(* Logix 5000 project; controller APM Emulate 5570 rev 30.12; software revision 30.00 *)

TASK MainTask (continuous, watchdog 500 ms) : MainProgram

MODULES
   Local : Emulate 5570 (ICP 2, rev 30.12)
      I_O1 : vendor 1 type 0 code 15 (ICP 3, rev 1.1, Output RPI 150 ms)
      I_O2 : vendor 1 type 0 code 15 (ICP 4, rev 1.1, Output RPI 150 ms)
END_MODULES

PROGRAM MainProgram   (* main routine MainRoutine *)
VAR
   CT_ACT_C050 : BOOL;
   CT_ACT_C051 : BOOL;
   CT_ACT_C052 : BOOL;
   CT_ACT_C053 : BOOL;
   CT_ACT_C054 : BOOL;
   CT_ACT_C055 : BOOL;
   CT_ACT_C056 : BOOL;
   CT_ACT_C260 : BOOL;
   CT_ACT_C261 : BOOL;
   CT_ACT_C262 : BOOL;
   CT_ACT_C263 : BOOL;
   CT_ACT_C264 : BOOL;
   CT_ACT_C265 : BOOL;
   CT_ACT_C266 : BOOL;
   CT_ACT_HOM : BOOL;
   CT_ACT_MSP0 : BOOL;
   CT_ACT_MSP1 : BOOL;
   CT_ACT_STP : BOOL;
   CT_ACT_VER0 : BOOL;
   CT_ACT_VER1 : BOOL;
   CT_ACT_VER2 : BOOL;
   CT_CA_AVC : BOOL;
   CT_CA_RET : BOOL;
   CT_CC_AVC : BOOL;
   CT_CC_RET : BOOL;
   CT_CP_AVC : BOOL;
   CT_CP_RET : BOOL;
   CT_DIS : INT;
   CT_OK : BOOL;
   CT_PBT_ESTP : ALIAS FOR Local:4:I.Data[1].0;
   CT_PBT_STA : ALIAS FOR Local:4:I.Data[1].1;
   CT_PBT_STP : ALIAS FOR Local:4:I.Data[1].2;
   CT_SEN_AAV : ALIAS FOR Local:4:I.Data[1].4;
   CT_SEN_ARE : ALIAS FOR Local:4:I.Data[1].3;
   CT_SEN_CAV : ALIAS FOR Local:4:I.Data[1].6;
   CT_SEN_CRE : ALIAS FOR Local:4:I.Data[1].5;
   CT_SEN_M05 : ALIAS FOR Local:4:I.Data[1].11;
   CT_SEN_M26 : ALIAS FOR Local:4:I.Data[1].12;
   CT_SEN_MAT : ALIAS FOR Local:4:I.Data[1].9;
   CT_SEN_PAV : ALIAS FOR Local:4:I.Data[1].8;
   CT_SEN_PRE : ALIAS FOR Local:4:I.Data[1].7;
   CT_SEQ_C05 : BOOL;
   CT_SEQ_C26 : BOOL;
   CT_SEQ_MSP : BOOL;
   CT_SEQ_VER : BOOL;
   MAIN_ACTIVE : BOOL;
   MAIN_PBT_ESTP : ALIAS FOR Local:3:I.Data[1].0;
   MAIN_PBT_STA : ALIAS FOR Local:3:I.Data[1].1;
   PNT_ACT_0 : BOOL;
   PNT_ACT_1 : BOOL;
   PNT_ACT_2 : BOOL;
   PNT_ACT_3 : BOOL;
   PNT_ACT_4 : BOOL;
   PNT_ACT_HOM : BOOL;
   PNT_MTA_AVC : BOOL;
   PNT_MTA_RET : BOOL;
   PNT_MTA_STP : BOOL;
   PNT_MTB_AVC : BOOL;
   PNT_MTB_RET : BOOL;
   PNT_MTB_STP : BOOL;
   PNT_MTC_AVC : BOOL;
   PNT_MTC_RET : BOOL;
   PNT_MTC_STP : BOOL;
   PNT_PBT_HOM : ALIAS FOR Local:3:I.Data[1].10;
   PNT_PBT_STA : ALIAS FOR Local:3:I.Data[1].11;
   PNT_PBT_STP : ALIAS FOR Local:3:I.Data[1].12;
   PNT_SEN_1 : ALIAS FOR Local:3:I.Data[1].13;
   PNT_SEN_2 : ALIAS FOR Local:3:I.Data[1].14;
   PNT_SEN_3 : ALIAS FOR Local:3:I.Data[1].15;
   PNT_SEN_4 : ALIAS FOR Local:3:I.Data[1].16;
   PNT_SEN_5 : ALIAS FOR Local:3:I.Data[1].17;
   PNT_SEN_6 : ALIAS FOR Local:3:I.Data[1].18;
   PNT_SEN_7 : ALIAS FOR Local:3:I.Data[1].19;
   PNT_TM1 : TIMER := (PRE := 2000);
   test : BOOL;
END_VAR

ROUTINE Corte_actions   (* ladder *)
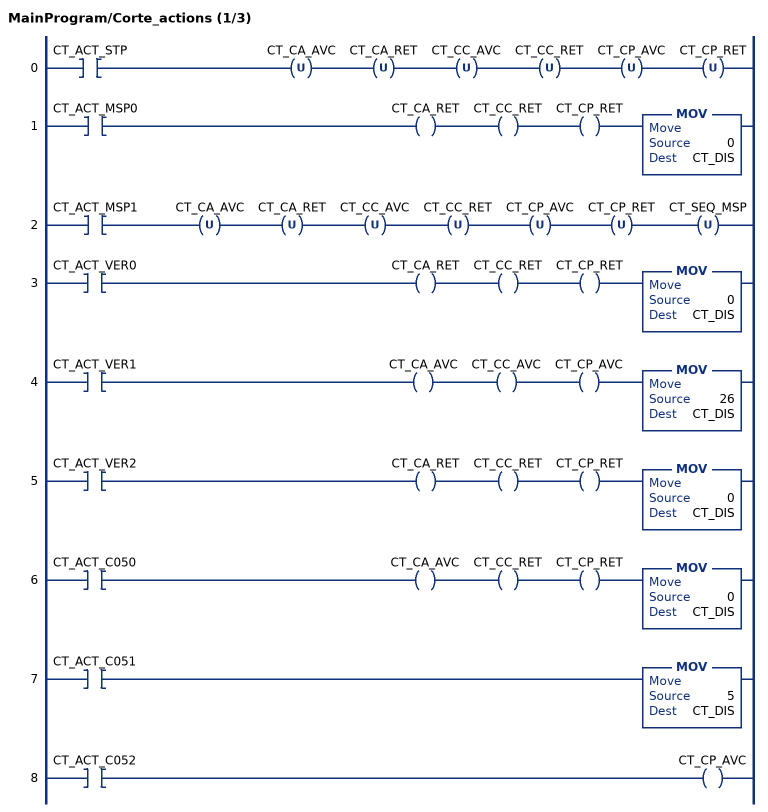
   0: XIC(CT_ACT_STP)OTU(CT_CA_AVC)OTU(CT_CA_RET)OTU(CT_CC_AVC)OTU(CT_CC_RET)OTU(CT_CP_AVC)OTU(CT_CP_RET);
   1: XIC(CT_ACT_MSP0)OTE(CT_CA_RET)OTE(CT_CC_RET)OTE(CT_CP_RET)MOV(0,CT_DIS);
   2: XIC(CT_ACT_MSP1)OTU(CT_CA_AVC)OTU(CT_CA_RET)OTU(CT_CC_AVC)OTU(CT_CC_RET)OTU(CT_CP_AVC)OTU(CT_CP_RET)OTU(CT_SEQ_MSP);
   3: XIC(CT_ACT_VER0)OTE(CT_CA_RET)OTE(CT_CC_RET)OTE(CT_CP_RET)MOV(0,CT_DIS);
   4: XIC(CT_ACT_VER1)OTE(CT_CA_AVC)OTE(CT_CC_AVC)OTE(CT_CP_AVC)MOV(26,CT_DIS);
   5: XIC(CT_ACT_VER2)OTE(CT_CA_RET)OTE(CT_CC_RET)OTE(CT_CP_RET)MOV(0,CT_DIS);
   6: XIC(CT_ACT_C050)OTE(CT_CA_AVC)OTE(CT_CC_RET)OTE(CT_CP_RET)MOV(0,CT_DIS);
   7: XIC(CT_ACT_C051)MOV(5,CT_DIS);
   8: XIC(CT_ACT_C052)OTE(CT_CP_AVC);
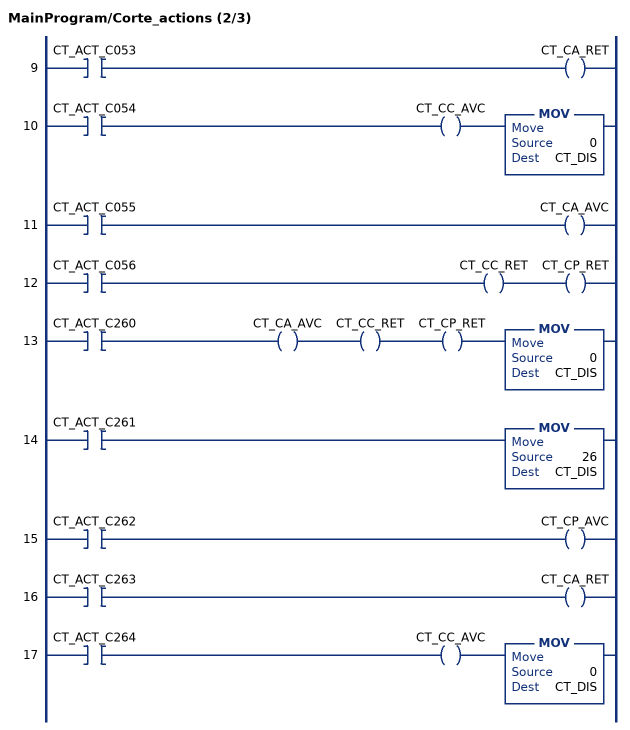
   9: XIC(CT_ACT_C053)OTE(CT_CA_RET);
   10: XIC(CT_ACT_C054)OTE(CT_CC_AVC)MOV(0,CT_DIS);
   11: XIC(CT_ACT_C055)OTE(CT_CA_AVC);
   12: XIC(CT_ACT_C056)OTE(CT_CC_RET)OTE(CT_CP_RET);
   13: XIC(CT_ACT_C260)OTE(CT_CA_AVC)OTE(CT_CC_RET)OTE(CT_CP_RET)MOV(0,CT_DIS);
   14: XIC(CT_ACT_C261)MOV(26,CT_DIS);
   15: XIC(CT_ACT_C262)OTE(CT_CP_AVC);
   16: XIC(CT_ACT_C263)OTE(CT_CA_RET);
   17: XIC(CT_ACT_C264)OTE(CT_CC_AVC)MOV(0,CT_DIS);
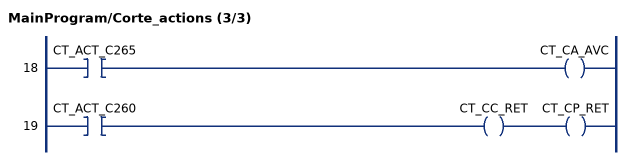
   18: XIC(CT_ACT_C265)OTE(CT_CA_AVC);
   19: XIC(CT_ACT_C260)OTE(CT_CC_RET)OTE(CT_CP_RET);
END_ROUTINE

ROUTINE Corte_logic   (* ladder *)
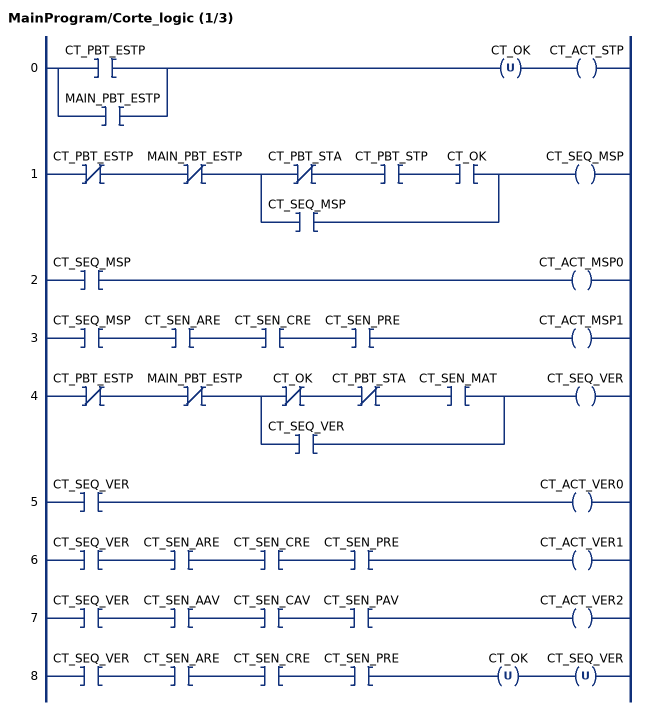
   0: [XIC(CT_PBT_ESTP) ,XIC(MAIN_PBT_ESTP) ]OTU(CT_OK)OTE(CT_ACT_STP);
   1: XIO(CT_PBT_ESTP)XIO(MAIN_PBT_ESTP)[XIO(CT_PBT_STA) XIC(CT_PBT_STP) XIC(CT_OK) ,XIC(CT_SEQ_MSP) ]OTE(CT_SEQ_MSP);
   2: XIC(CT_SEQ_MSP)OTE(CT_ACT_MSP0);
   3: XIC(CT_SEQ_MSP)XIC(CT_SEN_ARE)XIC(CT_SEN_CRE)XIC(CT_SEN_PRE)OTE(CT_ACT_MSP1);
   4: XIO(CT_PBT_ESTP)XIO(MAIN_PBT_ESTP)[XIO(CT_OK) XIO(CT_PBT_STA) XIC(CT_SEN_MAT) ,XIC(CT_SEQ_VER) ]OTE(CT_SEQ_VER);
   5: XIC(CT_SEQ_VER)OTE(CT_ACT_VER0);
   6: XIC(CT_SEQ_VER)XIC(CT_SEN_ARE)XIC(CT_SEN_CRE)XIC(CT_SEN_PRE)OTE(CT_ACT_VER1);
   7: XIC(CT_SEQ_VER)XIC(CT_SEN_AAV)XIC(CT_SEN_CAV)XIC(CT_SEN_PAV)OTE(CT_ACT_VER2);
   8: XIC(CT_SEQ_VER)XIC(CT_SEN_ARE)XIC(CT_SEN_CRE)XIC(CT_SEN_PRE)OTU(CT_OK)OTU(CT_SEQ_VER);
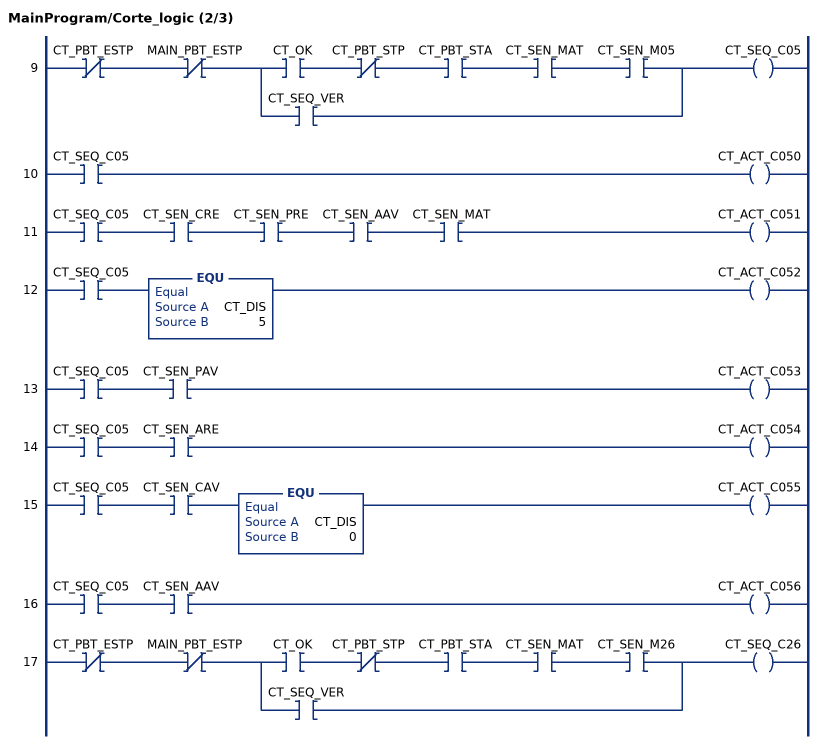
   9: XIO(CT_PBT_ESTP)XIO(MAIN_PBT_ESTP)[XIC(CT_OK) XIO(CT_PBT_STP) XIC(CT_PBT_STA) XIC(CT_SEN_MAT) XIC(CT_SEN_M05) ,XIC(CT_SEQ_VER) ]OTE(CT_SEQ_C05);
   10: XIC(CT_SEQ_C05)OTE(CT_ACT_C050);
   11: XIC(CT_SEQ_C05)XIC(CT_SEN_CRE)XIC(CT_SEN_PRE)XIC(CT_SEN_AAV)XIC(CT_SEN_MAT)OTE(CT_ACT_C051);
   12: XIC(CT_SEQ_C05)EQU(CT_DIS,5)OTE(CT_ACT_C052);
   13: XIC(CT_SEQ_C05)XIC(CT_SEN_PAV)OTE(CT_ACT_C053);
   14: XIC(CT_SEQ_C05)XIC(CT_SEN_ARE)OTE(CT_ACT_C054);
   15: XIC(CT_SEQ_C05)XIC(CT_SEN_CAV)EQU(CT_DIS,0)OTE(CT_ACT_C055);
   16: XIC(CT_SEQ_C05)XIC(CT_SEN_AAV)OTE(CT_ACT_C056);
   17: XIO(CT_PBT_ESTP)XIO(MAIN_PBT_ESTP)[XIC(CT_OK) XIO(CT_PBT_STP) XIC(CT_PBT_STA) XIC(CT_SEN_MAT) XIC(CT_SEN_M26) ,XIC(CT_SEQ_VER) ]OTE(CT_SEQ_C26);
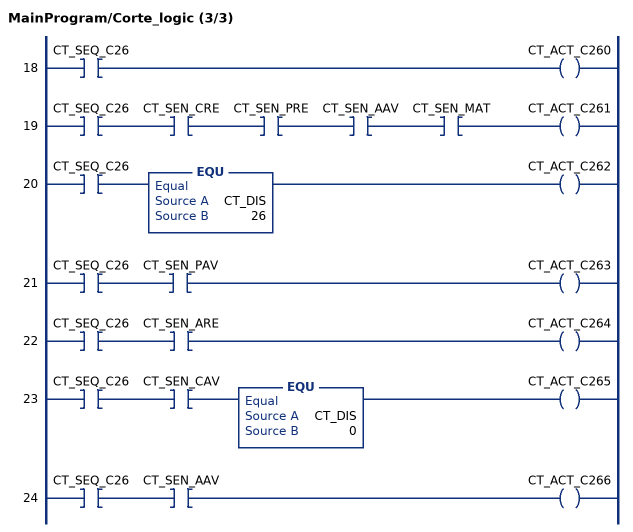
   18: XIC(CT_SEQ_C26)OTE(CT_ACT_C260);
   19: XIC(CT_SEQ_C26)XIC(CT_SEN_CRE)XIC(CT_SEN_PRE)XIC(CT_SEN_AAV)XIC(CT_SEN_MAT)OTE(CT_ACT_C261);
   20: XIC(CT_SEQ_C26)EQU(CT_DIS,26)OTE(CT_ACT_C262);
   21: XIC(CT_SEQ_C26)XIC(CT_SEN_PAV)OTE(CT_ACT_C263);
   22: XIC(CT_SEQ_C26)XIC(CT_SEN_ARE)OTE(CT_ACT_C264);
   23: XIC(CT_SEQ_C26)XIC(CT_SEN_CAV)EQU(CT_DIS,0)OTE(CT_ACT_C265);
   24: XIC(CT_SEQ_C26)XIC(CT_SEN_AAV)OTE(CT_ACT_C266);
END_ROUTINE

ROUTINE MainRoutine   (* ladder *)
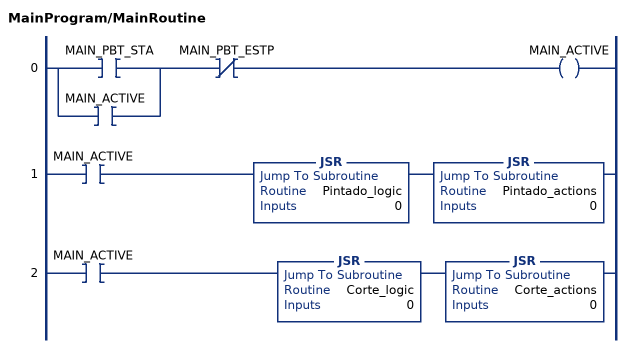
   0: [XIC(MAIN_PBT_STA) ,XIC(MAIN_ACTIVE) ]XIO(MAIN_PBT_ESTP)OTE(MAIN_ACTIVE);
   1: XIC(MAIN_ACTIVE)JSR(Pintado_logic,0)JSR(Pintado_actions,0);
   2: XIC(MAIN_ACTIVE)JSR(Corte_logic,0)JSR(Corte_actions,0);
END_ROUTINE

ROUTINE Pintado_actions   (* ladder *)
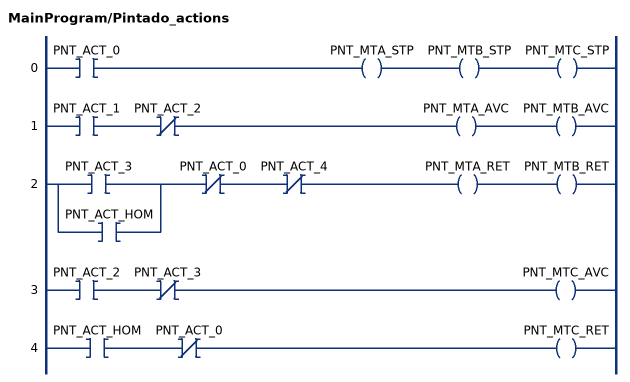
   0: XIC(PNT_ACT_0)OTE(PNT_MTA_STP)OTE(PNT_MTB_STP)OTE(PNT_MTC_STP);
   1: XIC(PNT_ACT_1)XIO(PNT_ACT_2)OTE(PNT_MTA_AVC)OTE(PNT_MTB_AVC);
   2: [XIC(PNT_ACT_3) ,XIC(PNT_ACT_HOM) ]XIO(PNT_ACT_0)XIO(PNT_ACT_4)OTE(PNT_MTA_RET)OTE(PNT_MTB_RET);
   3: XIC(PNT_ACT_2)XIO(PNT_ACT_3)OTE(PNT_MTC_AVC);
   4: XIC(PNT_ACT_HOM)XIO(PNT_ACT_0)OTE(PNT_MTC_RET);
END_ROUTINE

ROUTINE Pintado_logic   (* ladder *)
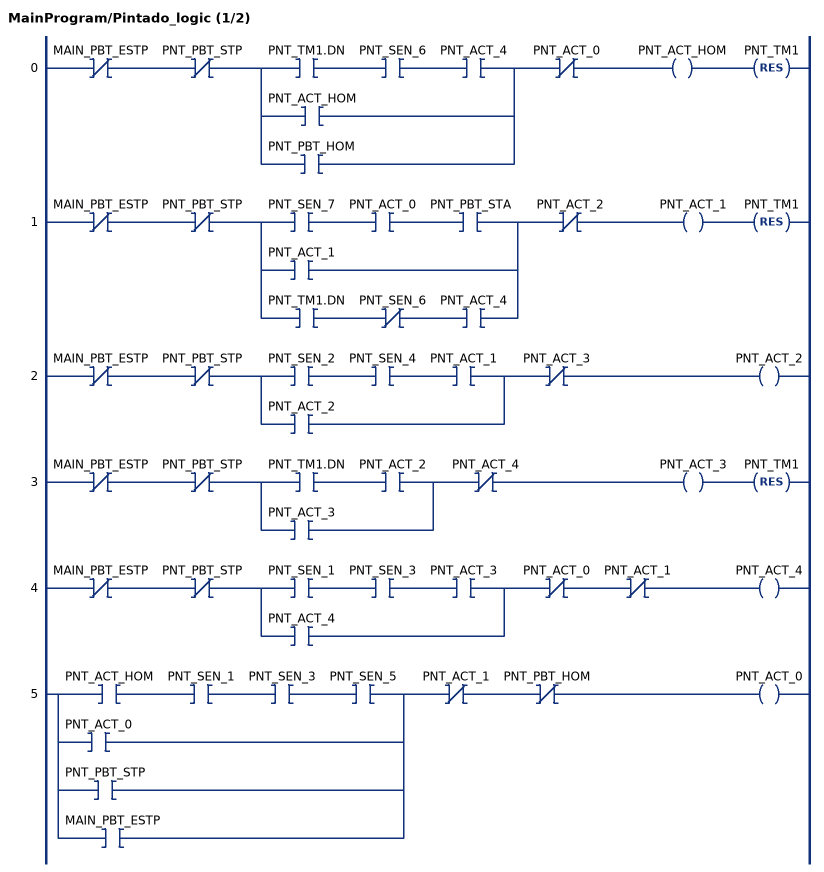
   0: XIO(MAIN_PBT_ESTP)XIO(PNT_PBT_STP)[XIC(PNT_TM1.DN) XIC(PNT_SEN_6) XIC(PNT_ACT_4) ,XIC(PNT_ACT_HOM) ,XIC(PNT_PBT_HOM) ]XIO(PNT_ACT_0)OTE(PNT_ACT_HOM)RES(PNT_TM1);
   1: XIO(MAIN_PBT_ESTP)XIO(PNT_PBT_STP)[XIC(PNT_SEN_7) XIC(PNT_ACT_0) XIC(PNT_PBT_STA) ,XIC(PNT_ACT_1) ,XIC(PNT_TM1.DN) XIO(PNT_SEN_6) XIC(PNT_ACT_4) ]XIO(PNT_ACT_2)OTE(PNT_ACT_1)RES(PNT_TM1);
   2: XIO(MAIN_PBT_ESTP)XIO(PNT_PBT_STP)[XIC(PNT_SEN_2) XIC(PNT_SEN_4) XIC(PNT_ACT_1) ,XIC(PNT_ACT_2) ]XIO(PNT_ACT_3)OTE(PNT_ACT_2);
   3: XIO(MAIN_PBT_ESTP)XIO(PNT_PBT_STP)[XIC(PNT_TM1.DN) XIC(PNT_ACT_2) ,XIC(PNT_ACT_3) ]XIO(PNT_ACT_4)OTE(PNT_ACT_3)RES(PNT_TM1);
   4: XIO(MAIN_PBT_ESTP)XIO(PNT_PBT_STP)[XIC(PNT_SEN_1) XIC(PNT_SEN_3) XIC(PNT_ACT_3) ,XIC(PNT_ACT_4) ]XIO(PNT_ACT_0)XIO(PNT_ACT_1)OTE(PNT_ACT_4);
   5: [XIC(PNT_ACT_HOM) XIC(PNT_SEN_1) XIC(PNT_SEN_3) XIC(PNT_SEN_5) ,XIC(PNT_ACT_0) ,XIC(PNT_PBT_STP) ,XIC(MAIN_PBT_ESTP) ]XIO(PNT_ACT_1)XIO(PNT_PBT_HOM)OTE(PNT_ACT_0);
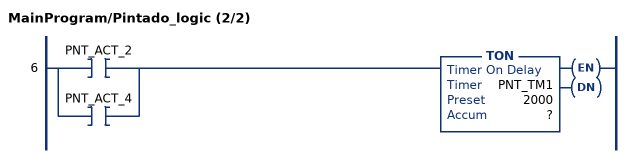
   6: [XIC(PNT_ACT_2) ,XIC(PNT_ACT_4) ]TON(PNT_TM1,?,?);
END_ROUTINE
END_PROGRAM
